TYPE ST_CAN_Frame :
STRUCT
    ID   : DWORD;                  // 29-bit CAN ID
    DLC  : BYTE;
    Data : ARRAY[0..7] OF BYTE;
END_STRUCT
END_TYPE

(* stored: Version 1.1.0.1, ProductVersion 3.1.4024.12
   DUT ST_CAN_Frame: Id {9def8077-7862-4204-8976-e693d35aafb1} *)
